INTERFACE I_Layers EXTENDS I_Object

{attribute 'OPC.UA.DA.Property' := '1'}
{attribute 'monitoring' := 'call'}
PROPERTY PUBLIC P_E0 : I_Layer
GET
END_GET
END_PROPERTY

{attribute 'OPC.UA.DA.Property' := '1'}
{attribute 'monitoring' := 'call'}
PROPERTY PUBLIC P_E1 : I_Layer
GET
END_GET
END_PROPERTY

{attribute 'OPC.UA.DA.Property' := '1'}
{attribute 'monitoring' := 'call'}
PROPERTY PUBLIC P_On : I_Layer
GET
END_GET
END_PROPERTY

END_INTERFACE

(* stored: Version 1.1.0.1
   Itf I_Layers: Id {c25d17bd-79d2-0c01-1bff-15c903946bd5}
   Property P_E0: Id {4fbbf462-1a1f-022a-344a-b813d786433d}
   Get Get: Id {a585f37d-ddfa-0f98-3177-f3da0ccda2a5}
   Property P_E1: Id {520ebbbb-8c71-0cf0-3a85-f6582e75d41d}
   Get Get: Id {085b248d-54d0-0011-1362-875d966eb670}
   Property P_On: Id {f4577bf3-23d3-0c41-1255-f02c5388499c}
   Get Get: Id {62b4361d-ec86-03f0-3695-ad875a1452d6} *)
